// TIA Portal V18 export
TYPE "MEStoPLC_MainCheckInStation2ST350_ext"
// stored: IsFailsafeCompliant false
   STRUCT
      PartTypeID : Int;   // Part type ID extracted from part type description
      Station1PalletID : Int;   // Pallet ID
      Station1PartSN : String[60];   // Serial number - Housing
      DataMatrixPartSN : String[60];   // 查询二维码
      Spare : Array[0..70] of Byte;   // 备用
      Massage : "MEStoPLC_AlarmMassage_ext";   // Process error code
   END_STRUCT;
END_TYPE
